TYPE I32 : DINT; END_TYPE

(* stored: Version 1.1.0.1
   DUT I32: Id {1b7bcae5-07c6-0129-315e-4fa0523b8a4c} *)
